// TIA Portal V15.1 export
// export: Created 2024-06-21T08:41:06.9518294Z, ExportSetting WithDefaults, DisplayName Totally Integrated Automation Portal, DisplayVersion V15.1 Update 5, DisplayName TIA Portal Openness, DisplayVersion V15.1 Update 5, DisplayName SINAMICS Startdrive Advanced, DisplayVersion V15.1, DisplayName G130, G150, S120, S150, SINAMICS MV, S210, DisplayVersion V15.1, DisplayName G110M, G120, G120C, G120D, G120P, DisplayVersion V15.1, DisplayName STEP 7 Professional, DisplayVersion V15.1 Update 5, DisplayName STEP 7 Safety, DisplayVersion V15.1, DisplayName WinCC Professional, DisplayVersion V15.1 Update 5, DisplayName SIMATIC Visualization Architect, DisplayVersion V15.1
FUNCTION_BLOCK "LGBProdSpeed"   // FB6699, FBD
TITLE = LGBProdSpeed
{ S7_Optimized_Access := 'TRUE' }
VERSION : 0.1
// stored: AutoNumber false, IsIECCheckEnabled false, IsRetainMemResEnabled false, MemoryReserve 100, SetENOAutomatically False, UDAEnableTagReadback false
   VAR_INPUT
      I_CRBodyPitch { ExternalAccessible := 'False'; ExternalVisible := 'False'; ExternalWritable := 'False'} : Int;   // Body pitch (cm) from control room
      I_CRCycleTime { ExternalAccessible := 'False'; ExternalVisible := 'False'; ExternalWritable := 'False'} : Int;   // Cycle time (sec) from control room
      I_CRSpeed { ExternalAccessible := 'False'; ExternalVisible := 'False'; ExternalWritable := 'False'} : Real;   // Speed (m/min) from control room
   END_VAR
   VAR_OUTPUT
      O_BodyPitch { ExternalAccessible := 'False'; ExternalVisible := 'False'; ExternalWritable := 'False'} : Int;   // Body pitch (cm)
      O_CycleTime { ExternalAccessible := 'False'; ExternalVisible := 'False'; ExternalWritable := 'False'} : Int;   // Cycle time (sec)
      "O_Speed(m/min)" { ExternalAccessible := 'False'; ExternalVisible := 'False'; ExternalWritable := 'False'} : Real;   // Speed (m/min)
      "O_Speed(mm/s)" { ExternalAccessible := 'False'; ExternalVisible := 'False'; ExternalWritable := 'False'} : Real;   // Speed (mm/s)
      O_AlarmABCondition { ExternalAccessible := 'False'; ExternalVisible := 'False'; ExternalWritable := 'False'} : Bool;   // Alarm AB Condition
      O_AlarmA { ExternalAccessible := 'False'; ExternalVisible := 'False'; ExternalWritable := 'False'} : Bool;   // Summation Alarm A of roller. / Alarm A
      O_AlarmB { ExternalAccessible := 'False'; ExternalVisible := 'False'; ExternalWritable := 'False'} : Bool;   // Summation Alarm B of roller. / Alarm B
      O_AlarmC { ExternalAccessible := 'False'; ExternalVisible := 'False'; ExternalWritable := 'False'} : Bool;   // Summation Alarm C of roller. / Alarm C
      O_AlarmD { ExternalAccessible := 'False'; ExternalVisible := 'False'; ExternalWritable := 'False'} : Bool;   // Summation Alarm D of roller. / Alarm D
      H_AlarmDWord { ExternalAccessible := 'False'; ExternalVisible := 'False'; ExternalWritable := 'False'} : DWord;   // Alarm Word
   END_VAR
   VAR_IN_OUT
      IO_Modes : "Modes";   // Modes
      H_HMI : "H_HMI";   // Animation
      H_GBProdSpeed : "H_GBProdSpeed";   // Animation
      C_Config : "ProdSpeedConfig";   // Config
   END_VAR
   VAR
      AC_CRBodyPitch { ExternalAccessible := 'False'; ExternalVisible := 'False'; ExternalWritable := 'False'} : Bool;   // The Body Pitch from control room is ZERO
      AC_CRCycleTime { ExternalAccessible := 'False'; ExternalVisible := 'False'; ExternalWritable := 'False'} : Bool;   // The Cycle Time from control room is ZERO
      AC_CRSpeed { ExternalAccessible := 'False'; ExternalVisible := 'False'; ExternalWritable := 'False'} : Bool;   // The Speed from control room is ZERO
      AC_LocalBodyPitch { ExternalAccessible := 'False'; ExternalVisible := 'False'; ExternalWritable := 'False'} : Bool;   // The local Body Pitch is ZERO
      AC_LocalCycleTime { ExternalAccessible := 'False'; ExternalVisible := 'False'; ExternalWritable := 'False'} : Bool;   // The lcoal Cycle Time is ZERO
      AC_LocalSpeed { ExternalAccessible := 'False'; ExternalVisible := 'False'; ExternalWritable := 'False'} : Bool;   // The local Speed is ZERO
      AC_CRLowestCycleTime { ExternalAccessible := 'False'; ExternalVisible := 'False'; ExternalWritable := 'False'} : Bool;   // The Cycle Time from control room is lower then the limit
      AC_CRHighestCycleTime { ExternalAccessible := 'False'; ExternalVisible := 'False'; ExternalWritable := 'False'} : Bool;   // The Cycle Time from control room is higher then the limit
      AC_LocalLowestCycleTime { ExternalAccessible := 'False'; ExternalVisible := 'False'; ExternalWritable := 'False'} : Bool;   // The local Cycle Time is lower then the limit
      AC_LocalHighestCycleTime { ExternalAccessible := 'False'; ExternalVisible := 'False'; ExternalWritable := 'False'} : Bool;   // The local Cycle Time is higher then the limit
      AD_Confirm { ExternalAccessible := 'False'; ExternalVisible := 'False'; ExternalWritable := 'False'} : Bool;   // The new setpoints are still not confirmed
      BodyPitch { ExternalAccessible := 'False'; ExternalVisible := 'False'; ExternalWritable := 'False'} : Int;   // Body pitch (cm)
      CycleTime { ExternalAccessible := 'False'; ExternalVisible := 'False'; ExternalWritable := 'False'} : Int;   // Cycle time (sec)
      Speed { ExternalAccessible := 'False'; ExternalVisible := 'False'; ExternalWritable := 'False'} : Real;   // Speed (m/min)
      LocalBodyPitch { ExternalAccessible := 'False'; ExternalVisible := 'False'; ExternalWritable := 'False'} : Int;   // Local Body pitch (cm)
      LocalCycleTime { ExternalAccessible := 'False'; ExternalVisible := 'False'; ExternalWritable := 'False'} : Int;   // Local Cycle time (sec)
      LocalSpeed { ExternalAccessible := 'False'; ExternalVisible := 'False'; ExternalWritable := 'False'} : Real;   // Local Speed (m/min)
      MemLocalBodyPitch { ExternalAccessible := 'False'; ExternalVisible := 'False'; ExternalWritable := 'False'} : Int;   // Memory Local Body pitch (cm)
      MemLocalCycleTime { ExternalAccessible := 'False'; ExternalVisible := 'False'; ExternalWritable := 'False'} : Int;   // Memory Local Cycle time (sec)
      MemLocalSpeed { ExternalAccessible := 'False'; ExternalVisible := 'False'; ExternalWritable := 'False'} : Real;   // Memory Local Speed (m/min)
      MemHMICMDSetpCR { ExternalAccessible := 'False'; ExternalVisible := 'False'; ExternalWritable := 'False'} : Bool;   // Memory HMI Command
      MemHMICMDSetpLocal { ExternalAccessible := 'False'; ExternalVisible := 'False'; ExternalWritable := 'False'} : Bool;   // Memory HMI Command
      Confirm { ExternalAccessible := 'False'; ExternalVisible := 'False'; ExternalWritable := 'False'} : Bool;   // Confirm new settings
      AlarmA { ExternalAccessible := 'False'; ExternalVisible := 'False'; ExternalWritable := 'False'} : Bool;   // Summation Alarm A of roller. / Alarm A / AlarmA
      AlarmB { ExternalAccessible := 'False'; ExternalVisible := 'False'; ExternalWritable := 'False'} : Bool;   // Summation Alarm B of roller. / Alarm B / AlarmB
      AlarmC { ExternalAccessible := 'False'; ExternalVisible := 'False'; ExternalWritable := 'False'} : Bool;   // Summation Alarm C of roller. / Alarm C / AlarmC
      AlarmD { ExternalAccessible := 'False'; ExternalVisible := 'False'; ExternalWritable := 'False'} : Bool;   // Summation Alarm D of roller. / Alarm D / AlarmD
      AlarmABCondition { ExternalAccessible := 'False'; ExternalVisible := 'False'; ExternalWritable := 'False'} : Bool;   // Alarm AB Condition
      Alarm { ExternalAccessible := 'False'; ExternalVisible := 'False'; ExternalWritable := 'False'} : Bool;   // Alarm AB
      TimerConfirm { ExternalAccessible := 'False'; ExternalVisible := 'False'; ExternalWritable := 'False'} : TON_TIME;   // Timer
      Edge { ExternalAccessible := 'False'; ExternalVisible := 'False'; ExternalWritable := 'False'} : Array[0..10] of Bool;   // Edge
      HMICMD { ExternalAccessible := 'False'; ExternalVisible := 'False'; ExternalWritable := 'False'} : Struct   // Temp / HMI commands
         SetpCR { ExternalAccessible := 'False'; ExternalVisible := 'False'; ExternalWritable := 'False'} : Bool;   // Setpoints from Control Room
         SetpLocal { ExternalAccessible := 'False'; ExternalVisible := 'False'; ExternalWritable := 'False'} : Bool;   // Setpoints Local
         Confirm { ExternalAccessible := 'False'; ExternalVisible := 'False'; ExternalWritable := 'False'} : Bool;   // Confirm
         "Btn50%" { ExternalAccessible := 'False'; ExternalVisible := 'False'; ExternalWritable := 'False'} : Bool;   // Button 50% production speed
         Spare4 { ExternalAccessible := 'False'; ExternalVisible := 'False'; ExternalWritable := 'False'} : Bool;   // Spare
         Spare5 { ExternalAccessible := 'False'; ExternalVisible := 'False'; ExternalWritable := 'False'} : Bool;   // Spare
         Spare6 { ExternalAccessible := 'False'; ExternalVisible := 'False'; ExternalWritable := 'False'} : Bool;   // Spare
         Spare7 { ExternalAccessible := 'False'; ExternalVisible := 'False'; ExternalWritable := 'False'} : Bool;   // Spare
         Spare8 { ExternalAccessible := 'False'; ExternalVisible := 'False'; ExternalWritable := 'False'} : Bool;   // Spare
         Spare9 { ExternalAccessible := 'False'; ExternalVisible := 'False'; ExternalWritable := 'False'} : Bool;   // Spare
         Spare10 { ExternalAccessible := 'False'; ExternalVisible := 'False'; ExternalWritable := 'False'} : Bool;   // Spare
         Spare11 { ExternalAccessible := 'False'; ExternalVisible := 'False'; ExternalWritable := 'False'} : Bool;   // Spare
         Spare12 { ExternalAccessible := 'False'; ExternalVisible := 'False'; ExternalWritable := 'False'} : Bool;   // Spare
         Spare13 { ExternalAccessible := 'False'; ExternalVisible := 'False'; ExternalWritable := 'False'} : Bool;   // Spare
         Spare14 { ExternalAccessible := 'False'; ExternalVisible := 'False'; ExternalWritable := 'False'} : Bool;   // Spare
         Spare15 { ExternalAccessible := 'False'; ExternalVisible := 'False'; ExternalWritable := 'False'} : Bool;   // Spare
         Spare16 { ExternalAccessible := 'False'; ExternalVisible := 'False'; ExternalWritable := 'False'} : Bool;   // Spare
         Spare17 { ExternalAccessible := 'False'; ExternalVisible := 'False'; ExternalWritable := 'False'} : Bool;   // Spare
         Spare18 { ExternalAccessible := 'False'; ExternalVisible := 'False'; ExternalWritable := 'False'} : Bool;   // Spare
         Spare19 { ExternalAccessible := 'False'; ExternalVisible := 'False'; ExternalWritable := 'False'} : Bool;   // Spare
         Spare20 { ExternalAccessible := 'False'; ExternalVisible := 'False'; ExternalWritable := 'False'} : Bool;   // Spare
         Spare21 { ExternalAccessible := 'False'; ExternalVisible := 'False'; ExternalWritable := 'False'} : Bool;   // Spare
         Spare22 { ExternalAccessible := 'False'; ExternalVisible := 'False'; ExternalWritable := 'False'} : Bool;   // Spare
         Spare23 { ExternalAccessible := 'False'; ExternalVisible := 'False'; ExternalWritable := 'False'} : Bool;   // Spare
         Spare24 { ExternalAccessible := 'False'; ExternalVisible := 'False'; ExternalWritable := 'False'} : Bool;   // Spare
         Spare25 { ExternalAccessible := 'False'; ExternalVisible := 'False'; ExternalWritable := 'False'} : Bool;   // Spare
         Spare26 { ExternalAccessible := 'False'; ExternalVisible := 'False'; ExternalWritable := 'False'} : Bool;   // Spare
         Spare27 { ExternalAccessible := 'False'; ExternalVisible := 'False'; ExternalWritable := 'False'} : Bool;   // Spare
         Spare28 { ExternalAccessible := 'False'; ExternalVisible := 'False'; ExternalWritable := 'False'} : Bool;   // Spare
         Spare29 { ExternalAccessible := 'False'; ExternalVisible := 'False'; ExternalWritable := 'False'} : Bool;   // Spare
         Spare30 { ExternalAccessible := 'False'; ExternalVisible := 'False'; ExternalWritable := 'False'} : Bool;   // Spare
         Spare31 { ExternalAccessible := 'False'; ExternalVisible := 'False'; ExternalWritable := 'False'} : Bool;   // Spare
      END_STRUCT;
      TempReal1 { ExternalAccessible := 'False'; ExternalVisible := 'False'; ExternalWritable := 'False'} : Real;   // Temp Value
      TempReal2 { ExternalAccessible := 'False'; ExternalVisible := 'False'; ExternalWritable := 'False'} : Real;   // Temp Value
      TempReal3 { ExternalAccessible := 'False'; ExternalVisible := 'False'; ExternalWritable := 'False'} : Real;   // Temp Value
      TempBodyPitch { ExternalAccessible := 'False'; ExternalVisible := 'False'; ExternalWritable := 'False'} : Real;   // Temp Value
      TempCycleTime { ExternalAccessible := 'False'; ExternalVisible := 'False'; ExternalWritable := 'False'} : Real;   // Temp Value
   END_VAR
   VAR_TEMP   // added for the SCL form of the ladder/FBD networks
      _w1 : Bool;
      _w2 : Bool;
      _w3 : Bool;
      _w4 : Bool;
   END_VAR
BEGIN

REGION Network 1: **** 1 - Inputs **** HMI Commands
   // HMI Commands
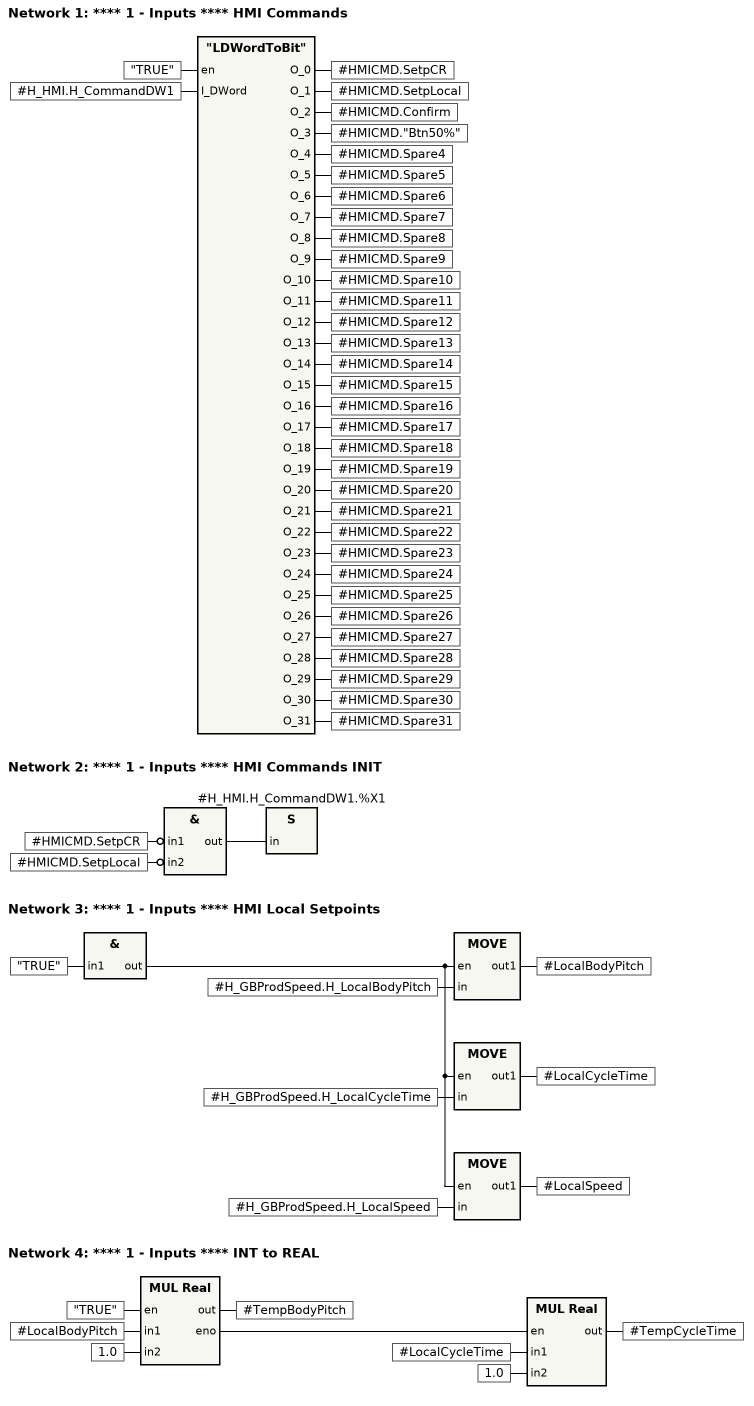
   IF "TRUE" THEN
       "LDWordToBit"(I_DWord := #H_HMI.H_CommandDW1,
                     O_0 => #HMICMD.SetpCR,
                     O_1 => #HMICMD.SetpLocal,
                     O_2 => #HMICMD.Confirm,
                     O_3 => #HMICMD."Btn50%",
                     O_4 => #HMICMD.Spare4,
                     O_5 => #HMICMD.Spare5,
                     O_6 => #HMICMD.Spare6,
                     O_7 => #HMICMD.Spare7,
                     O_8 => #HMICMD.Spare8,
                     O_9 => #HMICMD.Spare9,
                     O_10 => #HMICMD.Spare10,
                     O_11 => #HMICMD.Spare11,
                     O_12 => #HMICMD.Spare12,
                     O_13 => #HMICMD.Spare13,
                     O_14 => #HMICMD.Spare14,
                     O_15 => #HMICMD.Spare15,
                     O_16 => #HMICMD.Spare16,
                     O_17 => #HMICMD.Spare17,
                     O_18 => #HMICMD.Spare18,
                     O_19 => #HMICMD.Spare19,
                     O_20 => #HMICMD.Spare20,
                     O_21 => #HMICMD.Spare21,
                     O_22 => #HMICMD.Spare22,
                     O_23 => #HMICMD.Spare23,
                     O_24 => #HMICMD.Spare24,
                     O_25 => #HMICMD.Spare25,
                     O_26 => #HMICMD.Spare26,
                     O_27 => #HMICMD.Spare27,
                     O_28 => #HMICMD.Spare28,
                     O_29 => #HMICMD.Spare29,
                     O_30 => #HMICMD.Spare30,
                     O_31 => #HMICMD.Spare31);
   END_IF;
END_REGION

REGION Network 2: **** 1 - Inputs **** HMI Commands INIT
   IF NOT #HMICMD.SetpCR AND NOT #HMICMD.SetpLocal THEN #H_HMI.H_CommandDW1.%X1 := TRUE; END_IF;
END_REGION

REGION Network 3: **** 1 - Inputs **** HMI Local Setpoints
   IF "TRUE" THEN
       #LocalBodyPitch := #H_GBProdSpeed.H_LocalBodyPitch;
       #LocalCycleTime := #H_GBProdSpeed.H_LocalCycleTime;
       #LocalSpeed := #H_GBProdSpeed.H_LocalSpeed;
   END_IF;
END_REGION

REGION Network 4: **** 1 - Inputs **** INT to REAL
   IF "TRUE" THEN
       #TempBodyPitch := #LocalBodyPitch * 1.0;
       #TempCycleTime := #LocalCycleTime * 1.0;
   END_IF;
END_REGION

REGION Network 5: **** 2.2 - Alarms - Alarms Generation **** The Body Pitch from control room is ZERO
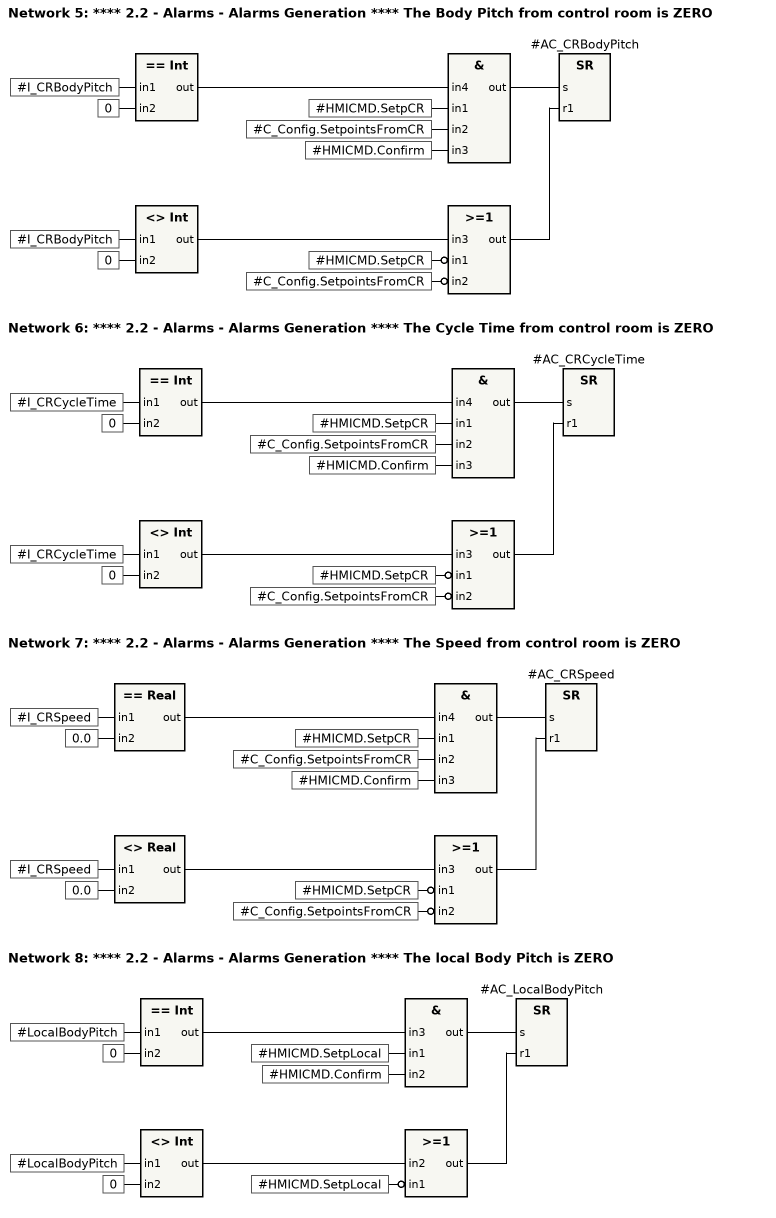
   IF (#I_CRBodyPitch = 0) AND #HMICMD.SetpCR AND #C_Config.SetpointsFromCR AND #HMICMD.Confirm THEN
       #AC_CRBodyPitch := TRUE;   // SR flip-flop
   END_IF;
   IF (#I_CRBodyPitch <> 0) OR NOT #HMICMD.SetpCR OR NOT #C_Config.SetpointsFromCR THEN
       #AC_CRBodyPitch := FALSE;
   END_IF;
END_REGION

REGION Network 6: **** 2.2 - Alarms - Alarms Generation **** The Cycle Time from control room is ZERO
   IF (#I_CRCycleTime = 0) AND #HMICMD.SetpCR AND #C_Config.SetpointsFromCR AND #HMICMD.Confirm THEN
       #AC_CRCycleTime := TRUE;   // SR flip-flop
   END_IF;
   IF (#I_CRCycleTime <> 0) OR NOT #HMICMD.SetpCR OR NOT #C_Config.SetpointsFromCR THEN
       #AC_CRCycleTime := FALSE;
   END_IF;
END_REGION

REGION Network 7: **** 2.2 - Alarms - Alarms Generation **** The Speed from control room is ZERO
   IF (#I_CRSpeed = 0.0) AND #HMICMD.SetpCR AND #C_Config.SetpointsFromCR AND #HMICMD.Confirm THEN
       #AC_CRSpeed := TRUE;   // SR flip-flop
   END_IF;
   IF (#I_CRSpeed <> 0.0) OR NOT #HMICMD.SetpCR OR NOT #C_Config.SetpointsFromCR THEN
       #AC_CRSpeed := FALSE;
   END_IF;
END_REGION

REGION Network 8: **** 2.2 - Alarms - Alarms Generation **** The local Body Pitch is ZERO
   IF (#LocalBodyPitch = 0) AND #HMICMD.SetpLocal AND #HMICMD.Confirm THEN
       #AC_LocalBodyPitch := TRUE;   // SR flip-flop
   END_IF;
   IF (#LocalBodyPitch <> 0) OR NOT #HMICMD.SetpLocal THEN #AC_LocalBodyPitch := FALSE; END_IF;
END_REGION

REGION Network 9: **** 2.2 - Alarms - Alarms Generation **** The lcoal Cycle Time is ZERO
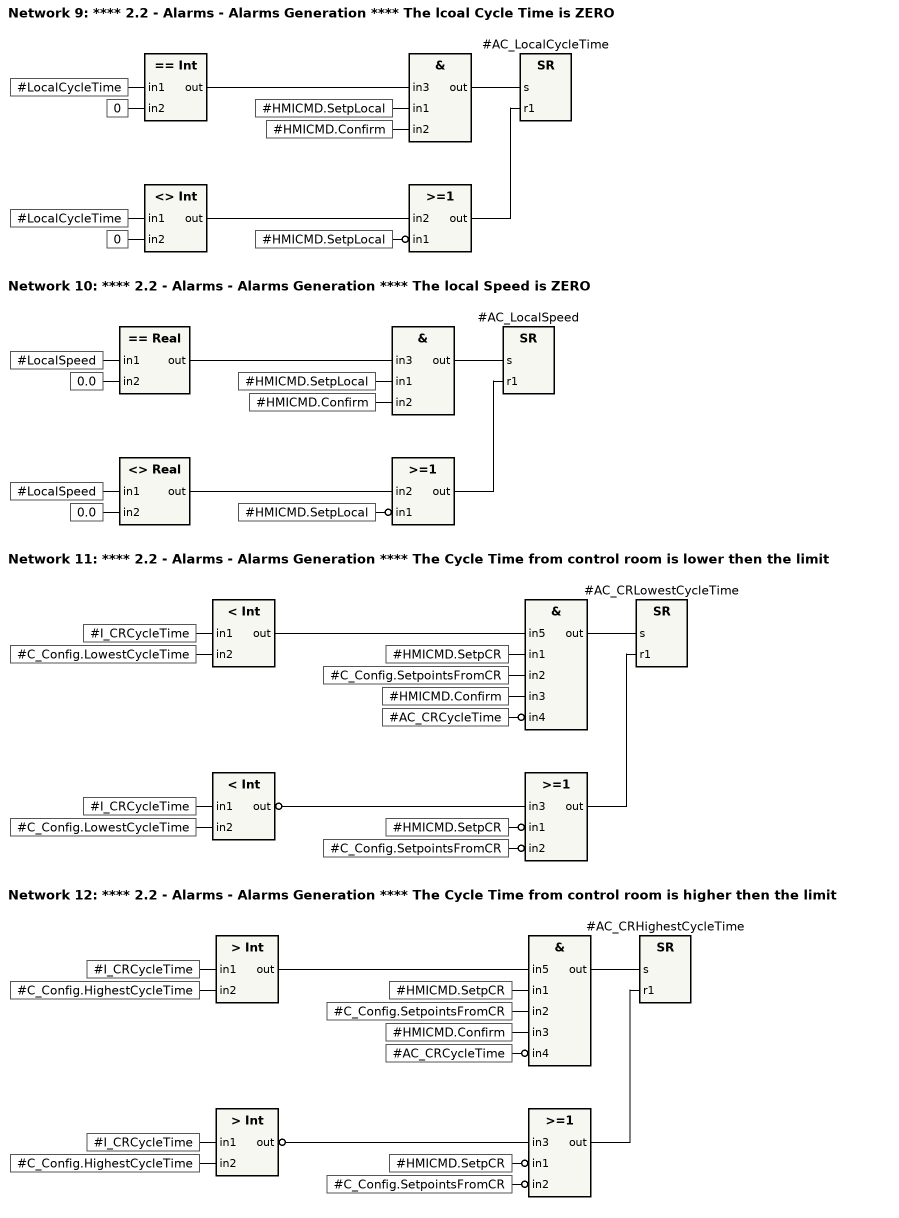
   IF (#LocalCycleTime = 0) AND #HMICMD.SetpLocal AND #HMICMD.Confirm THEN
       #AC_LocalCycleTime := TRUE;   // SR flip-flop
   END_IF;
   IF (#LocalCycleTime <> 0) OR NOT #HMICMD.SetpLocal THEN #AC_LocalCycleTime := FALSE; END_IF;
END_REGION

REGION Network 10: **** 2.2 - Alarms - Alarms Generation **** The local Speed is ZERO
   IF (#LocalSpeed = 0.0) AND #HMICMD.SetpLocal AND #HMICMD.Confirm THEN
       #AC_LocalSpeed := TRUE;   // SR flip-flop
   END_IF;
   IF (#LocalSpeed <> 0.0) OR NOT #HMICMD.SetpLocal THEN #AC_LocalSpeed := FALSE; END_IF;
END_REGION

REGION Network 11: **** 2.2 - Alarms - Alarms Generation **** The Cycle Time from control room is lower then the limit
   IF (#I_CRCycleTime < #C_Config.LowestCycleTime) AND #HMICMD.SetpCR AND #C_Config.SetpointsFromCR AND #HMICMD.Confirm AND NOT #AC_CRCycleTime THEN
       #AC_CRLowestCycleTime := TRUE;   // SR flip-flop
   END_IF;
   IF NOT (#I_CRCycleTime < #C_Config.LowestCycleTime) OR NOT #HMICMD.SetpCR OR NOT #C_Config.SetpointsFromCR THEN
       #AC_CRLowestCycleTime := FALSE;
   END_IF;
END_REGION

REGION Network 12: **** 2.2 - Alarms - Alarms Generation **** The Cycle Time from control room is higher then the limit
   IF (#I_CRCycleTime > #C_Config.HighestCycleTime) AND #HMICMD.SetpCR AND #C_Config.SetpointsFromCR AND #HMICMD.Confirm AND NOT #AC_CRCycleTime THEN
       #AC_CRHighestCycleTime := TRUE;   // SR flip-flop
   END_IF;
   IF NOT (#I_CRCycleTime > #C_Config.HighestCycleTime) OR NOT #HMICMD.SetpCR OR NOT #C_Config.SetpointsFromCR THEN
       #AC_CRHighestCycleTime := FALSE;
   END_IF;
END_REGION

REGION Network 13: **** 2.2 - Alarms - Alarms Generation **** The local Cycle Time is lower then the limit
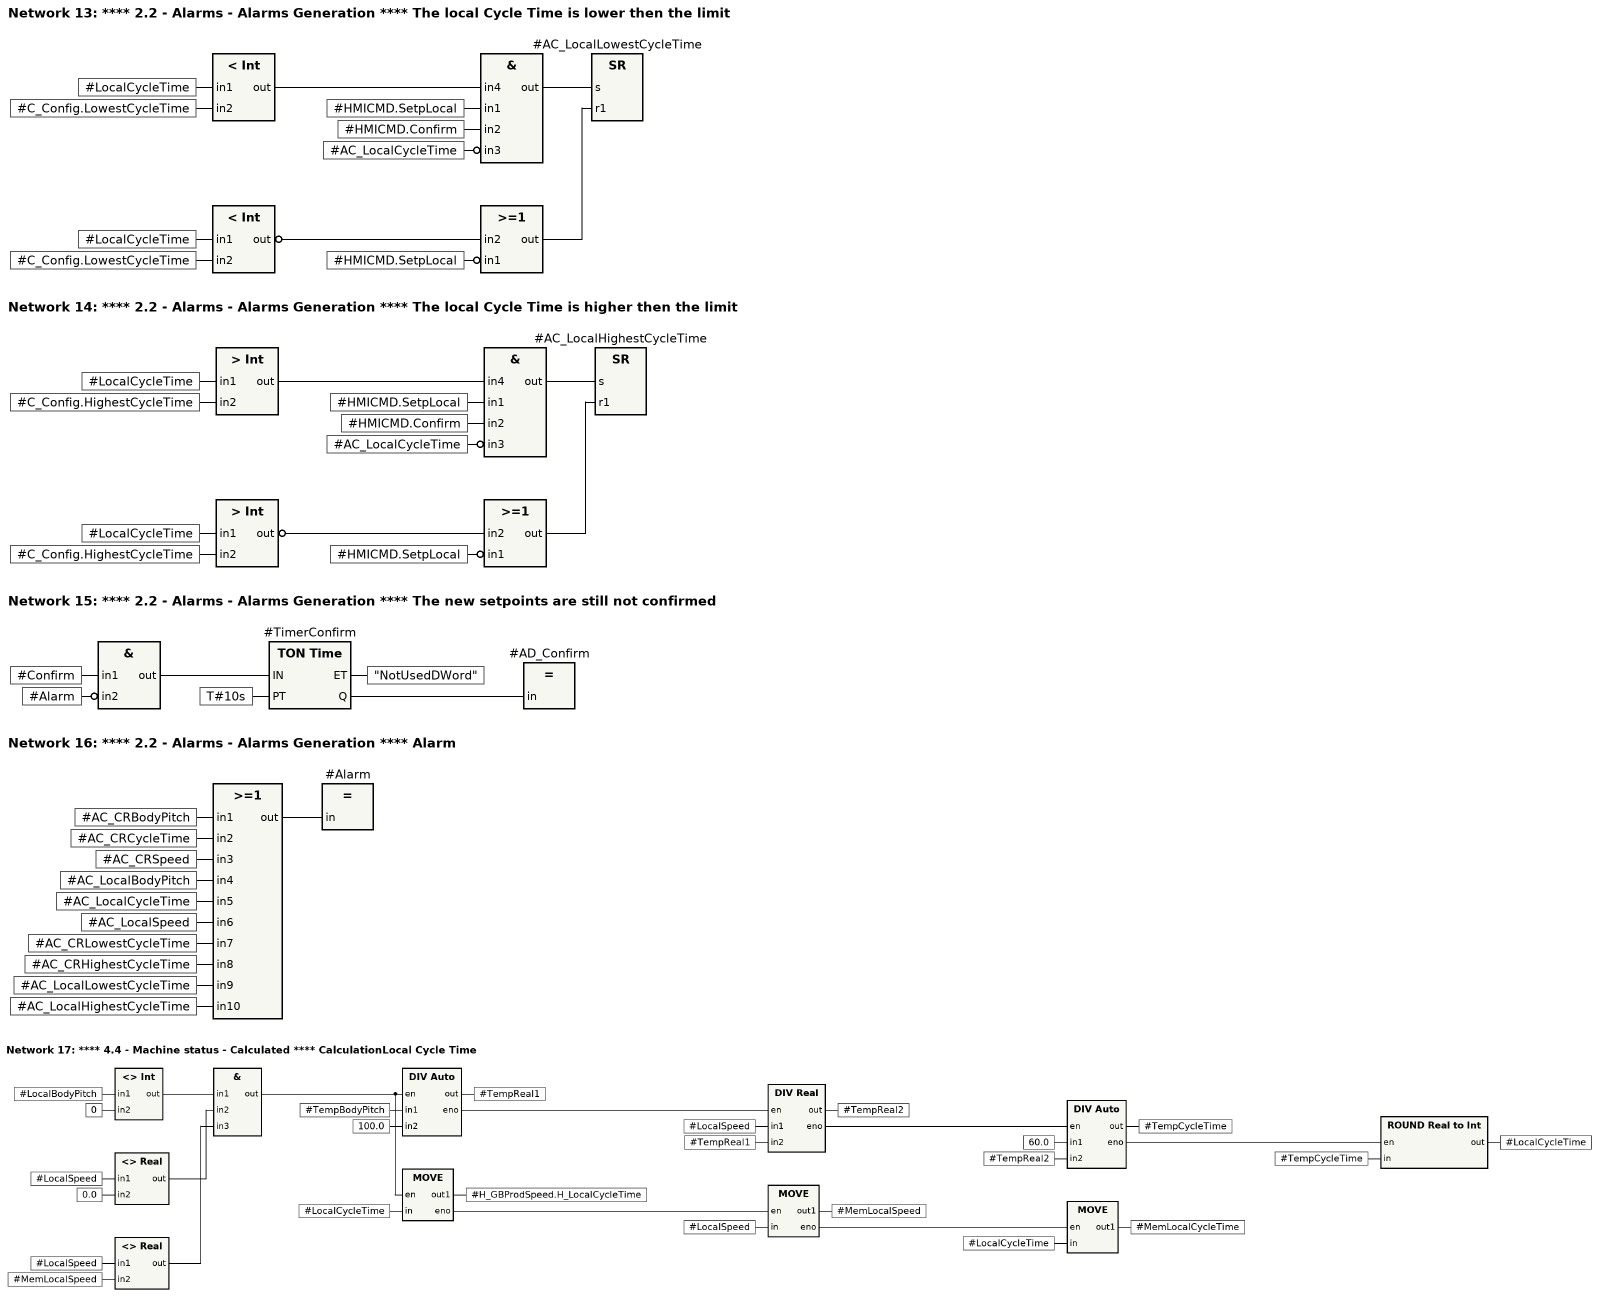
   IF (#LocalCycleTime < #C_Config.LowestCycleTime) AND #HMICMD.SetpLocal AND #HMICMD.Confirm AND NOT #AC_LocalCycleTime THEN
       #AC_LocalLowestCycleTime := TRUE;   // SR flip-flop
   END_IF;
   IF NOT (#LocalCycleTime < #C_Config.LowestCycleTime) OR NOT #HMICMD.SetpLocal THEN
       #AC_LocalLowestCycleTime := FALSE;
   END_IF;
END_REGION

REGION Network 14: **** 2.2 - Alarms - Alarms Generation **** The local Cycle Time is higher then the limit
   IF (#LocalCycleTime > #C_Config.HighestCycleTime) AND #HMICMD.SetpLocal AND #HMICMD.Confirm AND NOT #AC_LocalCycleTime THEN
       #AC_LocalHighestCycleTime := TRUE;   // SR flip-flop
   END_IF;
   IF NOT (#LocalCycleTime > #C_Config.HighestCycleTime) OR NOT #HMICMD.SetpLocal THEN
       #AC_LocalHighestCycleTime := FALSE;
   END_IF;
END_REGION

REGION Network 15: **** 2.2 - Alarms - Alarms Generation **** The new setpoints are still not confirmed
   #TimerConfirm(IN := #Confirm AND NOT #Alarm, PT := T#10s, ET => "NotUsedDWord");   // TON
   #AD_Confirm := #TimerConfirm.Q;
END_REGION

REGION Network 16: **** 2.2 - Alarms - Alarms Generation **** Alarm
   #Alarm := #AC_CRBodyPitch OR #AC_CRCycleTime OR #AC_CRSpeed OR #AC_LocalBodyPitch OR #AC_LocalCycleTime OR #AC_LocalSpeed OR #AC_CRLowestCycleTime OR #AC_CRHighestCycleTime OR #AC_LocalLowestCycleTime OR #AC_LocalHighestCycleTime;
END_REGION

REGION Network 17: **** 4.4 - Machine status - Calculated **** CalculationLocal Cycle Time
   IF (#LocalBodyPitch <> 0) AND (#LocalSpeed <> 0.0) AND (#LocalSpeed <> #MemLocalSpeed) THEN
       #TempReal1 := #TempBodyPitch / 100.0;
       #TempReal2 := #LocalSpeed / #TempReal1;
       #TempCycleTime := 60.0 / #TempReal2;
       #LocalCycleTime := ROUND(#TempCycleTime);
       #H_GBProdSpeed.H_LocalCycleTime := #LocalCycleTime;
   END_IF;
   #_w1 := (#LocalBodyPitch <> 0) AND (#LocalSpeed <> 0.0) AND (#LocalSpeed <> #MemLocalSpeed);
   IF #_w1 THEN
       #MemLocalSpeed := #LocalSpeed;
       #MemLocalCycleTime := #LocalCycleTime;
   END_IF;
END_REGION

REGION Network 18: **** 4.4 - Machine status - Calculated **** Calculation Local Speed
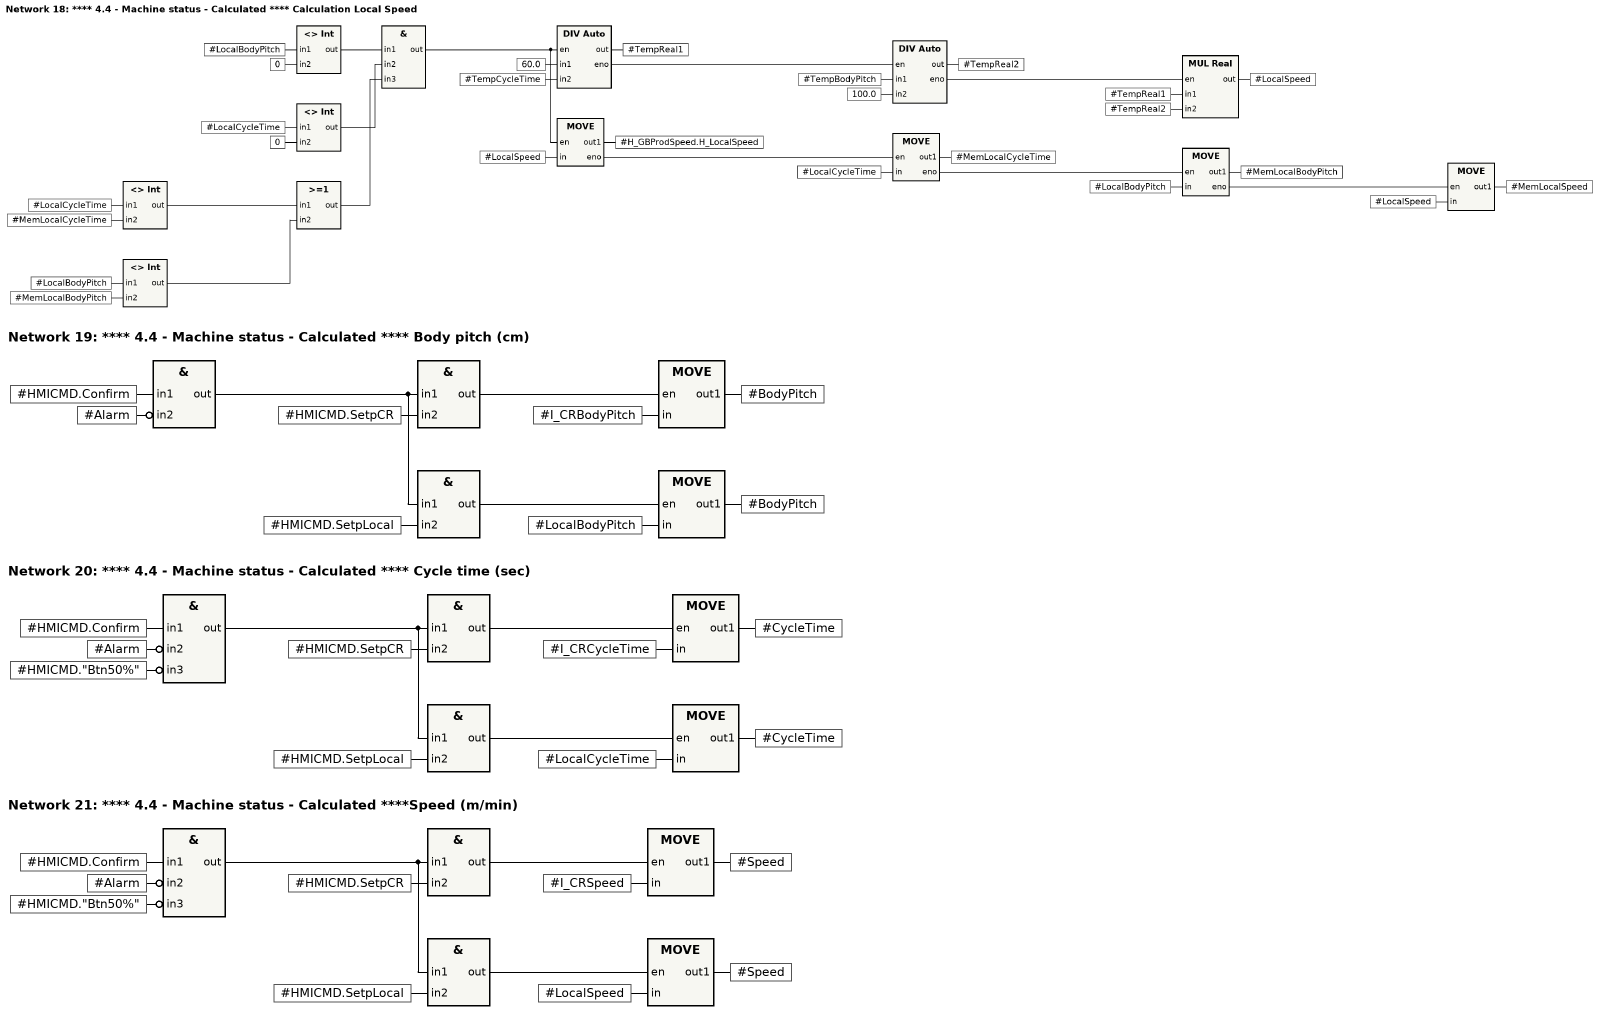
   IF (#LocalBodyPitch <> 0) AND (#LocalCycleTime <> 0) AND ((#LocalCycleTime <> #MemLocalCycleTime) OR (#LocalBodyPitch <> #MemLocalBodyPitch)) THEN
       #TempReal1 := 60.0 / #TempCycleTime;
       #TempReal2 := #TempBodyPitch / 100.0;
       #LocalSpeed := #TempReal1 * #TempReal2;
       #H_GBProdSpeed.H_LocalSpeed := #LocalSpeed;
   END_IF;
   #_w1 := (#LocalBodyPitch <> 0) AND (#LocalCycleTime <> 0) AND ((#LocalCycleTime <> #MemLocalCycleTime) OR (#LocalBodyPitch <> #MemLocalBodyPitch));
   IF #_w1 THEN
       #MemLocalCycleTime := #LocalCycleTime;
       #MemLocalBodyPitch := #LocalBodyPitch;
       #MemLocalSpeed := #LocalSpeed;
   END_IF;
END_REGION

REGION Network 19: **** 4.4 - Machine status - Calculated **** Body pitch (cm)
   #_w1 := #HMICMD.Confirm AND NOT #Alarm;
   IF #_w1 AND #HMICMD.SetpCR THEN #BodyPitch := #I_CRBodyPitch; END_IF;
   IF #_w1 AND #HMICMD.SetpLocal THEN #BodyPitch := #LocalBodyPitch; END_IF;
END_REGION

REGION Network 20: **** 4.4 - Machine status - Calculated **** Cycle time (sec)
   #_w1 := #HMICMD.Confirm AND NOT #Alarm AND NOT #HMICMD."Btn50%";
   IF #_w1 AND #HMICMD.SetpCR THEN #CycleTime := #I_CRCycleTime; END_IF;
   IF #_w1 AND #HMICMD.SetpLocal THEN #CycleTime := #LocalCycleTime; END_IF;
END_REGION

REGION Network 21: **** 4.4 - Machine status - Calculated ****Speed (m/min)
   #_w1 := #HMICMD.Confirm AND NOT #Alarm AND NOT #HMICMD."Btn50%";
   IF #_w1 AND #HMICMD.SetpCR THEN #Speed := #I_CRSpeed; END_IF;
   IF #_w1 AND #HMICMD.SetpLocal THEN #Speed := #LocalSpeed; END_IF;
END_REGION

REGION Network 22: **** 4.4 - Machine status - Calculated **** Button 50%
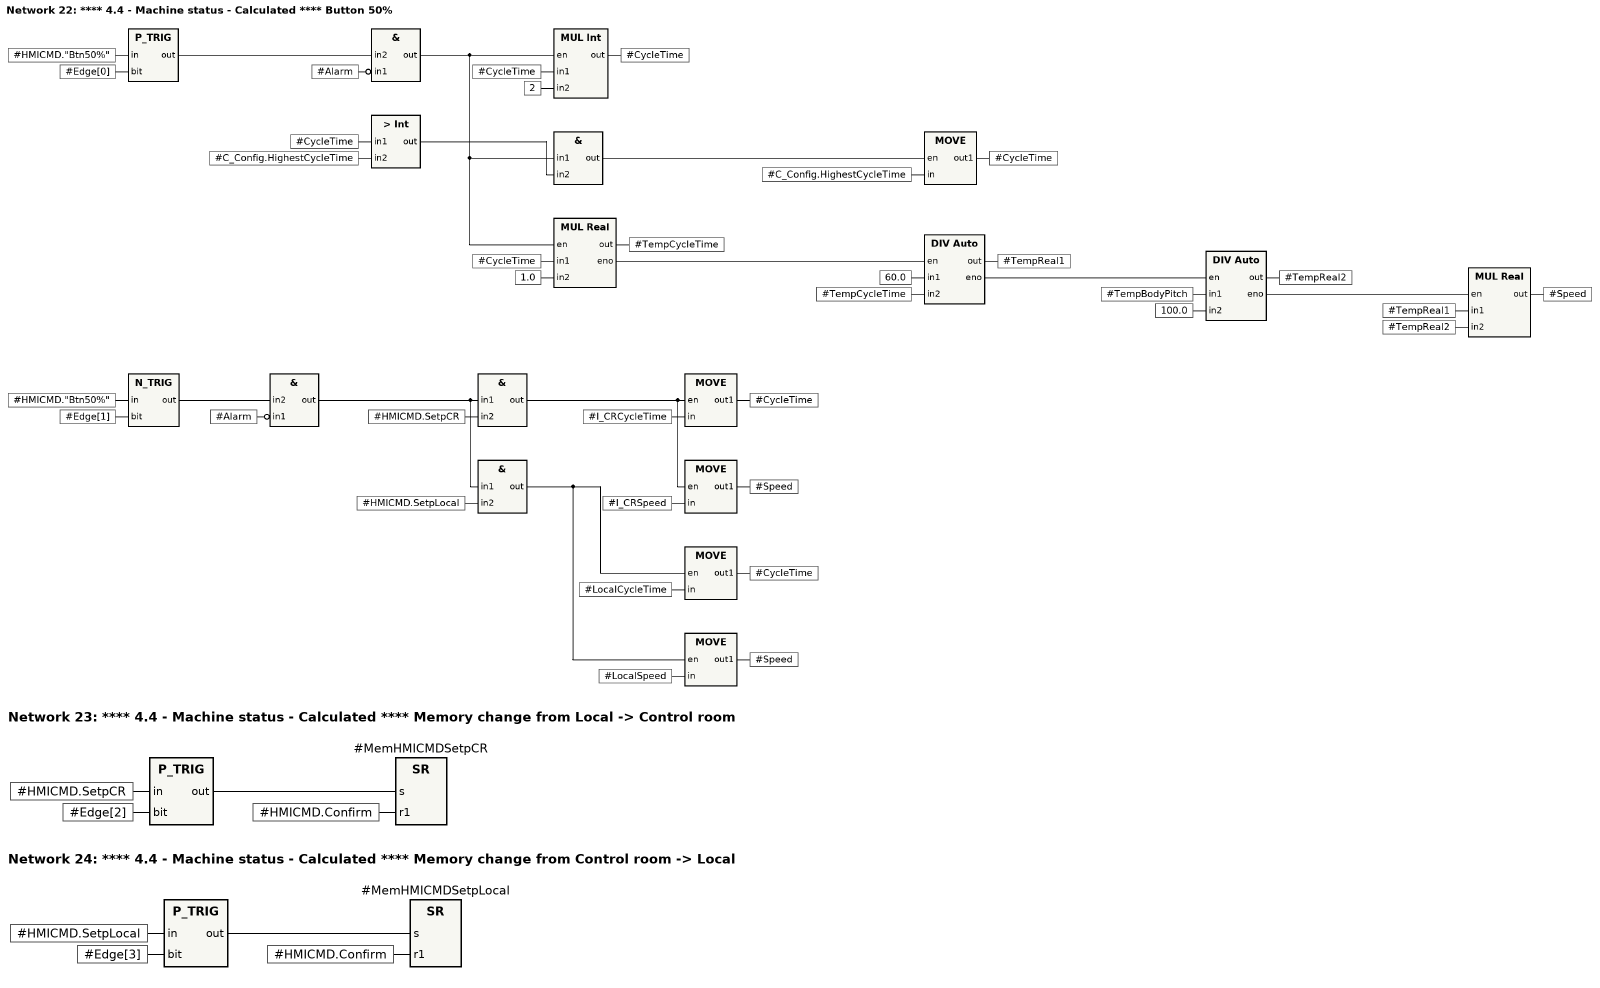
   #_w1 := #HMICMD."Btn50%" AND NOT #Edge[0];   // rising edge
   #Edge[0] := #HMICMD."Btn50%";
   #_w2 := #_w1 AND NOT #Alarm;
   IF #_w2 THEN #CycleTime := #CycleTime * 2; END_IF;
   IF #_w2 AND (#CycleTime > #C_Config.HighestCycleTime) THEN
       #CycleTime := #C_Config.HighestCycleTime;
   END_IF;
   IF #_w2 THEN
       #TempCycleTime := #CycleTime * 1.0;
       #TempReal1 := 60.0 / #TempCycleTime;
       #TempReal2 := #TempBodyPitch / 100.0;
       #Speed := #TempReal1 * #TempReal2;
   END_IF;
   #_w3 := NOT #HMICMD."Btn50%" AND #Edge[1];   // falling edge
   #Edge[1] := #HMICMD."Btn50%";
   #_w4 := #_w3 AND NOT #Alarm;
   IF #_w4 AND #HMICMD.SetpCR THEN
       #CycleTime := #I_CRCycleTime;
       #Speed := #I_CRSpeed;
   END_IF;
   IF #_w4 AND #HMICMD.SetpLocal THEN
       #CycleTime := #LocalCycleTime;
       #Speed := #LocalSpeed;
   END_IF;
END_REGION

REGION Network 23: **** 4.4 - Machine status - Calculated **** Memory change from Local -> Control room
   #_w1 := #HMICMD.SetpCR AND NOT #Edge[2];   // rising edge
   #Edge[2] := #HMICMD.SetpCR;
   IF #_w1 THEN
       #MemHMICMDSetpCR := TRUE;   // SR flip-flop
   END_IF;
   IF #HMICMD.Confirm THEN #MemHMICMDSetpCR := FALSE; END_IF;
END_REGION

REGION Network 24: **** 4.4 - Machine status - Calculated **** Memory change from Control room -> Local
   #_w1 := #HMICMD.SetpLocal AND NOT #Edge[3];   // rising edge
   #Edge[3] := #HMICMD.SetpLocal;
   IF #_w1 THEN
       #MemHMICMDSetpLocal := TRUE;   // SR flip-flop
   END_IF;
   IF #HMICMD.Confirm THEN #MemHMICMDSetpLocal := FALSE; END_IF;
END_REGION

REGION Network 25: **** 4.4 - Machine status - Calculated ****Confirm new setpoints
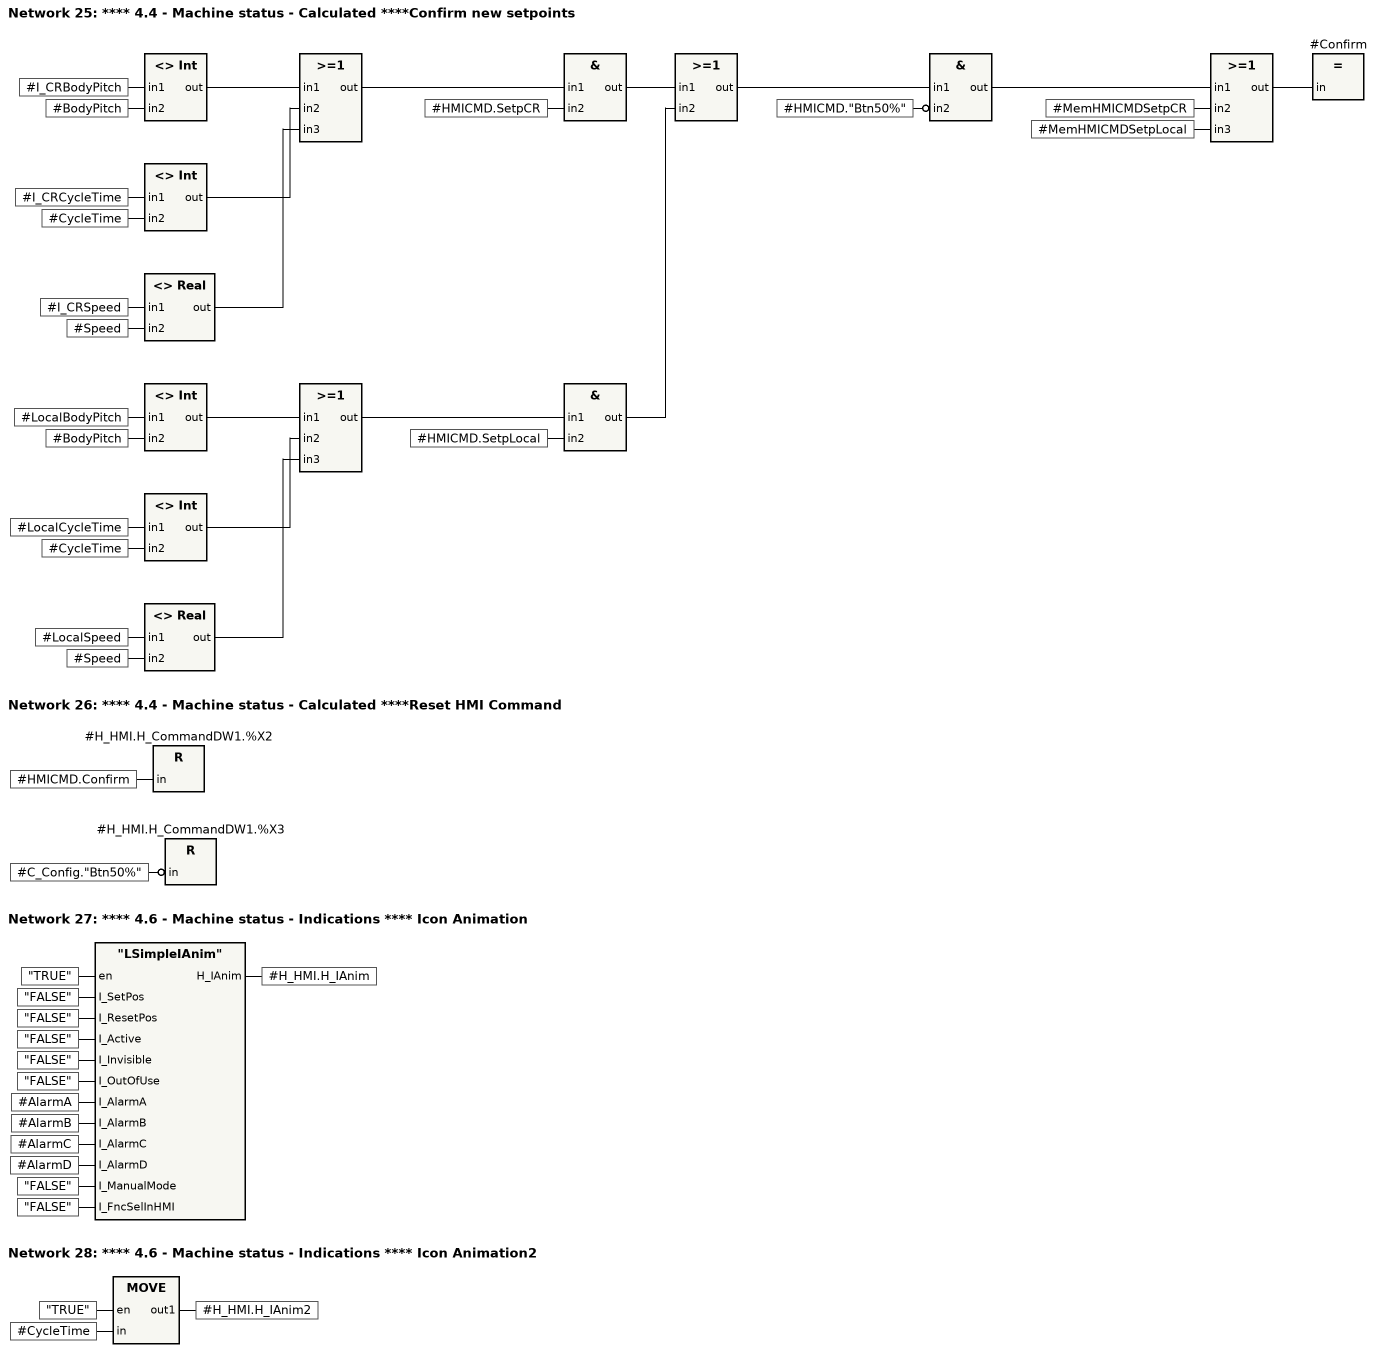
   #Confirm := (((((#I_CRBodyPitch <> #BodyPitch) OR (#I_CRCycleTime <> #CycleTime) OR (#I_CRSpeed <> #Speed)) AND #HMICMD.SetpCR) OR (((#LocalBodyPitch <> #BodyPitch) OR (#LocalCycleTime <> #CycleTime) OR (#LocalSpeed <> #Speed)) AND #HMICMD.SetpLocal)) AND NOT #HMICMD."Btn50%") OR #MemHMICMDSetpCR OR #MemHMICMDSetpLocal;
END_REGION

REGION Network 26: **** 4.4 - Machine status - Calculated ****Reset HMI Command
   IF #HMICMD.Confirm THEN #H_HMI.H_CommandDW1.%X2 := FALSE; END_IF;
   IF NOT #C_Config."Btn50%" THEN #H_HMI.H_CommandDW1.%X3 := FALSE; END_IF;
END_REGION

REGION Network 27: **** 4.6 - Machine status - Indications **** Icon Animation
   // Icon Animation for HMI
   IF "TRUE" THEN
       "LSimpleIAnim"(I_SetPos := "FALSE",
                      I_ResetPos := "FALSE",
                      I_Active := "FALSE",
                      I_Invisible := "FALSE",
                      I_OutOfUse := "FALSE",
                      I_AlarmA := #AlarmA,
                      I_AlarmB := #AlarmB,
                      I_AlarmC := #AlarmC,
                      I_AlarmD := #AlarmD,
                      I_ManualMode := "FALSE",
                      I_FncSelInHMI := "FALSE",
                      H_IAnim => #H_HMI.H_IAnim);
   END_IF;
END_REGION

REGION Network 28: **** 4.6 - Machine status - Indications **** Icon Animation2
   IF "TRUE" THEN #H_HMI.H_IAnim2 := #CycleTime; END_IF;
END_REGION

REGION Network 29: *** 4.6 - Machine Status - Indication **** Animation
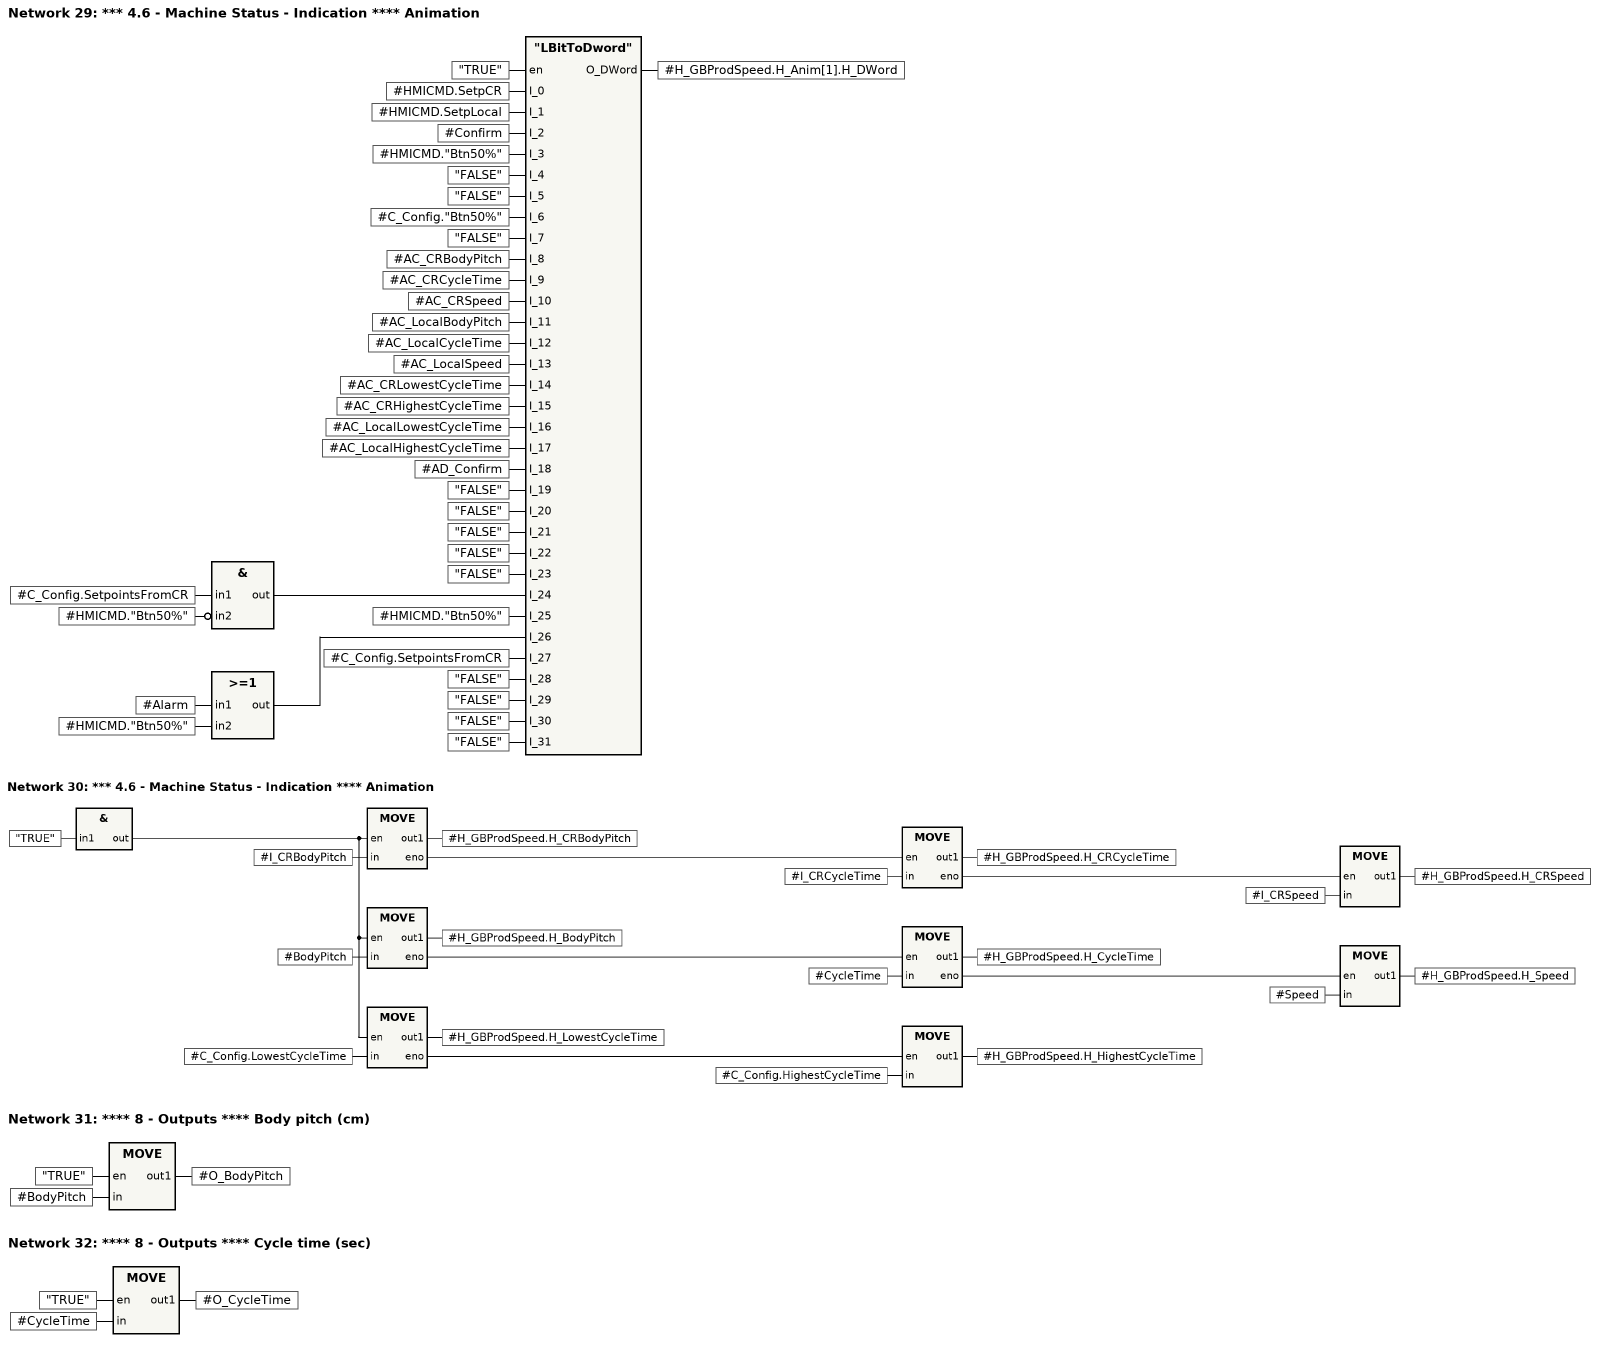
   IF "TRUE" THEN
       "LBitToDword"(I_0 := #HMICMD.SetpCR,
                     I_1 := #HMICMD.SetpLocal,
                     I_2 := #Confirm,
                     I_3 := #HMICMD."Btn50%",
                     I_4 := "FALSE",
                     I_5 := "FALSE",
                     I_6 := #C_Config."Btn50%",
                     I_7 := "FALSE",
                     I_8 := #AC_CRBodyPitch,
                     I_9 := #AC_CRCycleTime,
                     I_10 := #AC_CRSpeed,
                     I_11 := #AC_LocalBodyPitch,
                     I_12 := #AC_LocalCycleTime,
                     I_13 := #AC_LocalSpeed,
                     I_14 := #AC_CRLowestCycleTime,
                     I_15 := #AC_CRHighestCycleTime,
                     I_16 := #AC_LocalLowestCycleTime,
                     I_17 := #AC_LocalHighestCycleTime,
                     I_18 := #AD_Confirm,
                     I_19 := "FALSE",
                     I_20 := "FALSE",
                     I_21 := "FALSE",
                     I_22 := "FALSE",
                     I_23 := "FALSE",
                     I_24 := #C_Config.SetpointsFromCR AND NOT #HMICMD."Btn50%",
                     I_25 := #HMICMD."Btn50%",
                     I_26 := #Alarm OR #HMICMD."Btn50%",
                     I_27 := #C_Config.SetpointsFromCR,
                     I_28 := "FALSE",
                     I_29 := "FALSE",
                     I_30 := "FALSE",
                     I_31 := "FALSE",
                     O_DWord => #H_GBProdSpeed.H_Anim[1].H_DWord);
   END_IF;
END_REGION

REGION Network 30: *** 4.6 - Machine Status - Indication **** Animation
   IF "TRUE" THEN
       #H_GBProdSpeed.H_CRBodyPitch := #I_CRBodyPitch;
       #H_GBProdSpeed.H_CRCycleTime := #I_CRCycleTime;
       #H_GBProdSpeed.H_CRSpeed := #I_CRSpeed;
       #H_GBProdSpeed.H_BodyPitch := #BodyPitch;
       #H_GBProdSpeed.H_CycleTime := #CycleTime;
       #H_GBProdSpeed.H_Speed := #Speed;
       #H_GBProdSpeed.H_LowestCycleTime := #C_Config.LowestCycleTime;
       #H_GBProdSpeed.H_HighestCycleTime := #C_Config.HighestCycleTime;
   END_IF;
END_REGION

REGION Network 31: **** 8 - Outputs **** Body pitch (cm)
   IF "TRUE" THEN #O_BodyPitch := #BodyPitch; END_IF;
END_REGION

REGION Network 32: **** 8 - Outputs **** Cycle time (sec)
   IF "TRUE" THEN #O_CycleTime := #CycleTime; END_IF;
END_REGION

REGION Network 33: **** 8 - Outputs **** Speed (m/min)
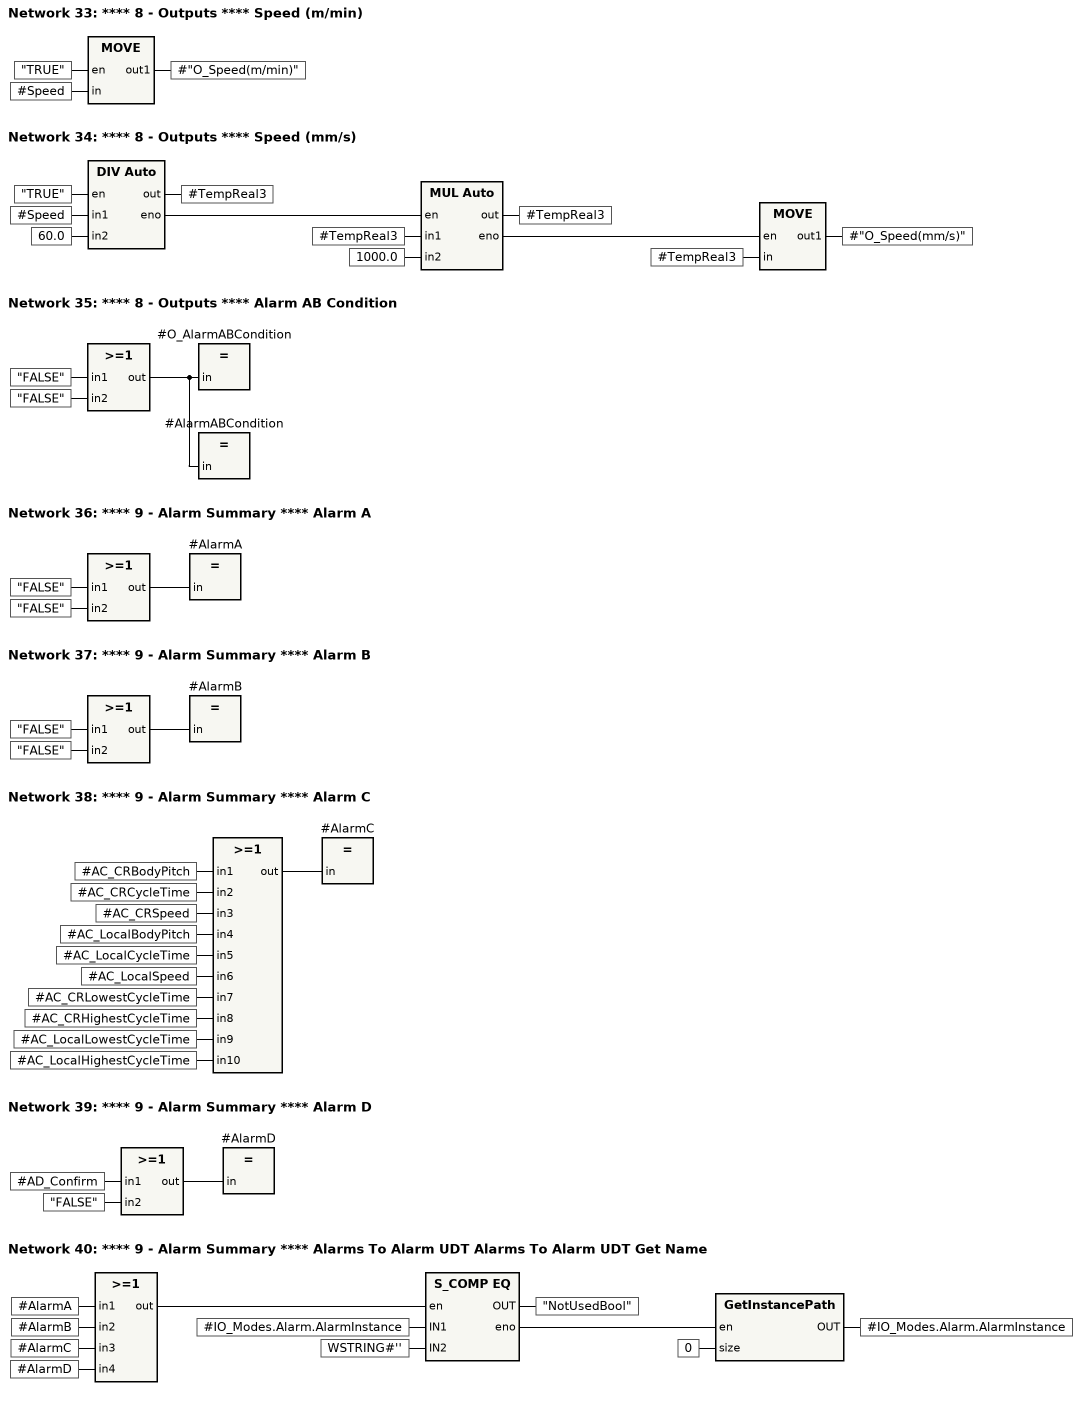
   IF "TRUE" THEN #"O_Speed(m/min)" := #Speed; END_IF;
END_REGION

REGION Network 34: **** 8 - Outputs **** Speed (mm/s)
   IF "TRUE" THEN
       #TempReal3 := #Speed / 60.0;
       #TempReal3 := #TempReal3 * 1000.0;
       #"O_Speed(mm/s)" := #TempReal3;
   END_IF;
END_REGION

REGION Network 35: **** 8 - Outputs **** Alarm AB Condition
   // Alarm AB Condition
   #O_AlarmABCondition := "FALSE" OR "FALSE";
   #AlarmABCondition := #O_AlarmABCondition;
END_REGION

REGION Network 36: **** 9 - Alarm Summary **** Alarm A
   // Alarm A
   #AlarmA := "FALSE" OR "FALSE";
END_REGION

REGION Network 37: **** 9 - Alarm Summary **** Alarm B
   // Alarm B
   #AlarmB := "FALSE" OR "FALSE";
END_REGION

REGION Network 38: **** 9 - Alarm Summary **** Alarm C
   // Alarm C
   #AlarmC := #AC_CRBodyPitch OR #AC_CRCycleTime OR #AC_CRSpeed OR #AC_LocalBodyPitch OR #AC_LocalCycleTime OR #AC_LocalSpeed OR #AC_CRLowestCycleTime OR #AC_CRHighestCycleTime OR #AC_LocalLowestCycleTime OR #AC_LocalHighestCycleTime;
END_REGION

REGION Network 39: **** 9 - Alarm Summary **** Alarm D
   // Alarm D
   #AlarmD := #AD_Confirm OR "FALSE";
END_REGION

REGION Network 40: **** 9 - Alarm Summary **** Alarms To Alarm UDT Alarms To Alarm UDT Get Name
   // Alarm / Alarm D
   S_COMP(EN := #AlarmA OR #AlarmB OR #AlarmC OR #AlarmD,
          IN1 := #IO_Modes.Alarm.AlarmInstance,
          IN2 := WSTRING#'',
          OUT => "NotUsedBool",
          ENO => #_w1);
   IF #_w1 THEN GetInstancePath(size := 0, OUT => #IO_Modes.Alarm.AlarmInstance); END_IF;
END_REGION

REGION Network 41: **** 9 - Alarm Summary **** Alarms To Alarm UDT
   // Alarm / Alarm D
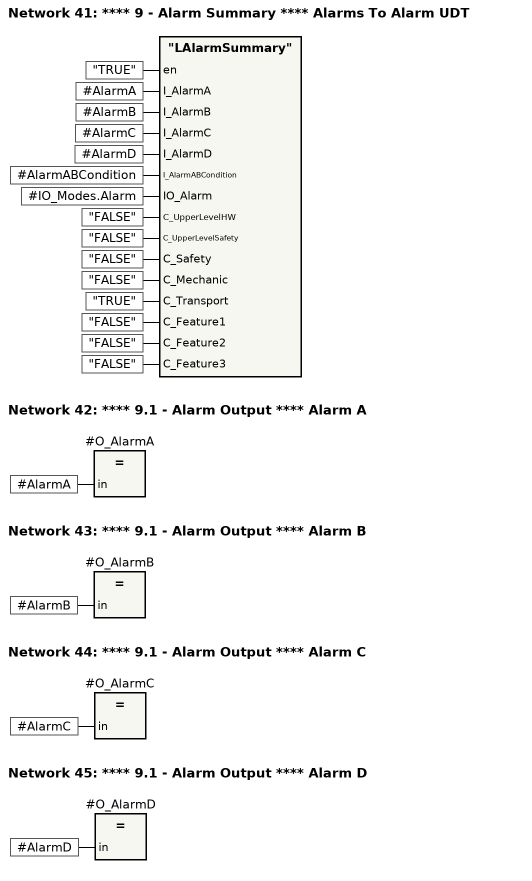
   IF "TRUE" THEN
       "LAlarmSummary"(I_AlarmA := #AlarmA,
                       I_AlarmB := #AlarmB,
                       I_AlarmC := #AlarmC,
                       I_AlarmD := #AlarmD,
                       I_AlarmABCondition := #AlarmABCondition,
                       IO_Alarm := #IO_Modes.Alarm,
                       C_UpperLevelHW := "FALSE",
                       C_UpperLevelSafety := "FALSE",
                       C_Safety := "FALSE",
                       C_Mechanic := "FALSE",
                       C_Transport := "TRUE",
                       C_Feature1 := "FALSE",
                       C_Feature2 := "FALSE",
                       C_Feature3 := "FALSE");
   END_IF;
END_REGION

REGION Network 42: **** 9.1 - Alarm Output **** Alarm A
   // Alarm A
   #O_AlarmA := #AlarmA;
END_REGION

REGION Network 43: **** 9.1 - Alarm Output **** Alarm B
   // Alarm B
   #O_AlarmB := #AlarmB;
END_REGION

REGION Network 44: **** 9.1 - Alarm Output **** Alarm C
   // Alarm C
   #O_AlarmC := #AlarmC;
END_REGION

REGION Network 45: **** 9.1 - Alarm Output **** Alarm D
   // Alarm D
   #O_AlarmD := #AlarmD;
END_REGION

REGION Network 46: **** 9.2 - Alarm DWord**** Alarm To DWord
   // Alarm To Word
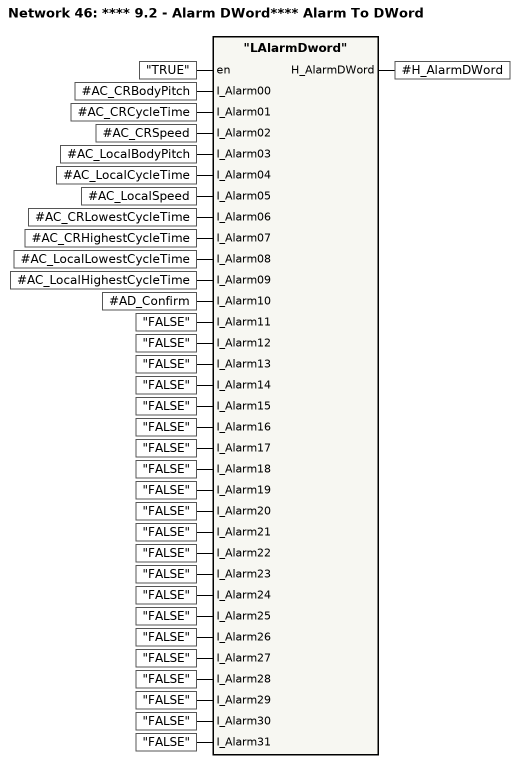
   IF "TRUE" THEN
       "LAlarmDword"(I_Alarm00 := #AC_CRBodyPitch,
                     I_Alarm01 := #AC_CRCycleTime,
                     I_Alarm02 := #AC_CRSpeed,
                     I_Alarm03 := #AC_LocalBodyPitch,
                     I_Alarm04 := #AC_LocalCycleTime,
                     I_Alarm05 := #AC_LocalSpeed,
                     I_Alarm06 := #AC_CRLowestCycleTime,
                     I_Alarm07 := #AC_CRHighestCycleTime,
                     I_Alarm08 := #AC_LocalLowestCycleTime,
                     I_Alarm09 := #AC_LocalHighestCycleTime,
                     I_Alarm10 := #AD_Confirm,
                     I_Alarm11 := "FALSE",
                     I_Alarm12 := "FALSE",
                     I_Alarm13 := "FALSE",
                     I_Alarm14 := "FALSE",
                     I_Alarm15 := "FALSE",
                     I_Alarm16 := "FALSE",
                     I_Alarm17 := "FALSE",
                     I_Alarm18 := "FALSE",
                     I_Alarm19 := "FALSE",
                     I_Alarm20 := "FALSE",
                     I_Alarm21 := "FALSE",
                     I_Alarm22 := "FALSE",
                     I_Alarm23 := "FALSE",
                     I_Alarm24 := "FALSE",
                     I_Alarm25 := "FALSE",
                     I_Alarm26 := "FALSE",
                     I_Alarm27 := "FALSE",
                     I_Alarm28 := "FALSE",
                     I_Alarm29 := "FALSE",
                     I_Alarm30 := "FALSE",
                     I_Alarm31 := "FALSE",
                     H_AlarmDWord => #H_AlarmDWord);
   END_IF;
END_REGION
END_FUNCTION_BLOCK
